// TIA Portal V19 export
TYPE "LEXCHANGETRAY_typeHandlingXyzEm_recieve_interface"
// stored: Access Published
   STRUCT
      constraintRoller { S7_SetPoint := 'True'} : "LEXCHANGETRAY_typeHandlingXyzEm_toConstraintRollerRecieve";
      plasticRoller { S7_SetPoint := 'True'} : "LEXCHANGETRAY_typeHandlingXyzEm_toPlasticRecieve";
      NgConvyorRoller { S7_SetPoint := 'True'} : "LEXCHANGETRAY_typeHandlingXyzEm_toNgConveyorRecieve";
   END_STRUCT;
END_TYPE
